// Mitsubishi GX Works2 project: 0709   PLC: Q02/Q02H

PROGRAM MAIN
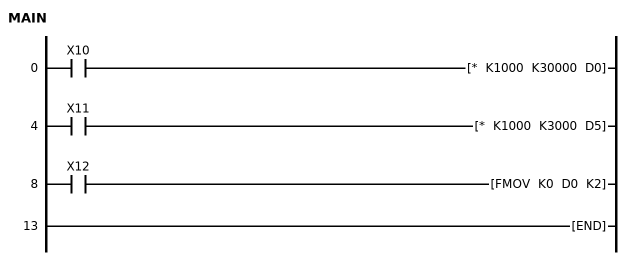
0     LD      X10
      *       K1000 K30000 D0
4     LD      X11
      *       K1000 K3000 D5
8     LD      X12
      FMOV    K0 D0 K2
13    END
END_PROGRAM
